PROGRAM MAIN
VAR
	fbAxis : FB_BaseAxis		(AxisName		:=	'Axis1',
								nPtpPoints		:=	5,
								iProcessHandler	:=	0,
								iTorqueLimiting	:=	0,
								iPosCamLookup	:=	0,
								iVeloCamLookup	:=	0,
								iPtpCamLookup	:=	0);
END_VAR

fbAxis();
MCgvl.fbMCOperationMode();

END_PROGRAM

(* stored: Version 1.1.0.1, ProductVersion 3.1.4024.6
   POU MAIN: Id {878ec357-822f-404b-844d-1b4014fa06cc}, SpecialFunc None *)
